TYPE ST_EVENT_DATA :
STRUCT
		String1: STRING;
		String2: STRING;
END_STRUCT
END_TYPE

(* stored: Version 1.1.0.1, ProductVersion 3.1.4024.12
   DUT ST_EVENT_DATA: Id {1939a44f-cdac-42f2-8225-a4c5950cfbc8} *)
